TYPE "ValveMachine_Manager"
VERSION : 0.1
// Block: ValveMachine_Manager
   STRUCT
      EnableStopDoorOpeningReq : Bool;
      EnableStopInPhase : Bool;
      EnableStopProgrammed : Bool;
      Control_ON : Bool;
      Rest : Bool;
      Work : Bool;
   END_STRUCT;

END_TYPE
